{attribute 'linkalways'} 
{attribute 'no_explicit_call' := 'This FB is a CLASS and must be accessed using methods or properties'}
{attribute 'enable_dynamic_creation'}
FUNCTION_BLOCK _DT EXTENDS DatatypeBase
VAR
	localData : DT;
	activeData : REFERENCE TO DT REF= localData;
END_VAR

PROPERTY PUBLIC Address : PVOID
GET
Address := ADR(activeData);
END_GET
END_PROPERTY

METHOD PUBLIC ClearReference
VAR_INPUT
END_VAR
activeData REF= localData;
END_METHOD

METHOD PUBLIC Clone : I_Datatype
VAR
    pClone : POINTER TO _DT;
END_VAR
pClone := __NEW(_DT(InitialValue := Value));
Clone := pClone^;
END_METHOD

METHOD FB_init : BOOL
VAR_INPUT
	bInitRetains : BOOL; // if TRUE, the retain variables are initialized (warm start / cold start)
	bInCopyCode : BOOL;  // if TRUE, the instance afterwards gets moved WORDo the copy code (online change)
	InitialValue : DT;
END_VAR
localData := InitialValue;
END_METHOD

PROPERTY PUBLIC IecType : T_MAXSTRING
GET
IecType := 'DT';
END_GET
END_PROPERTY

METHOD PUBLIC MakeReferenceTo
VAR_INPUT
	ReferenceTarget : REFERENCE TO DT;
END_VAR
activeData REF= ReferenceTarget;
END_METHOD

METHOD PUBLIC SerializeWith
VAR_INPUT
	Serializer : I_Serializer;
END_VAR
Serializer.AddDateTime(activeData);
END_METHOD

PROPERTY PUBLIC Size : UDINT
GET
Size := SIZEOF(activeData);
END_GET
END_PROPERTY

METHOD TryDeserializeFrom : BOOL
VAR_INPUT
	Deserializer : I_Deserializer;
	Feedback : I_DeserializerFeedback;
END_VAR
TryDeserializeFrom := Deserializer.TryGetDateTime(activeData, Feedback);
END_METHOD

METHOD TryMakeReferenceTo : BOOL
VAR_INPUT
	Target : I_Datatype;
END_VAR
VAR
	pTargetData : POINTER TO DT;
END_VAR
IF NOT (Target.IecType = IecType) THEN
	RETURN;
END_IF

pTargetData := Target.Address;
activeData REF= pTargetData^;
TryMakeReferenceTo := TRUE;
END_METHOD

PROPERTY PUBLIC Value : DT
GET
Value := activeData;
END_GET
SET
activeData := Value;
END_SET
END_PROPERTY

END_FUNCTION_BLOCK

(* stored: Version 1.1.0.1, ProductVersion 3.1.4024.12
   POU _DT: Id {5f0ed87a-efb3-0af3-3883-e19c081fdc00}, SpecialFunc None
   Folder Constructor: Id {29a57be8-9521-02ea-0210-43bf4e6f5595}
   Property Address: Id {01c07cd3-6ad8-0564-0c4b-2911104e3390}
   Get Get: Id {4c43ffa5-0c61-027d-3467-332c73ced3a6}
   Method ClearReference: Id {facc431e-3b24-02fc-2270-310f5a719454}
   Method Clone: Id {5f3d84b8-a743-0597-324d-f0078728fbc7}
   Method FB_init: Id {a1a061fc-f3bd-057e-3e6f-b4a094d0b439}
   Property IecType: Id {5a60c3be-49e4-0bea-33b1-0c3ea06f8245}
   Get Get: Id {0bd9b606-ce90-0f09-3b04-07eb42523072}
   Method MakeReferenceTo: Id {cfaca68c-b5d9-0493-2bd5-08d57f7cf5c8}
   Method SerializeWith: Id {058b9483-f6fd-0db0-2f66-9967c26a5006}
   Property Size: Id {cf76693d-be61-0e6e-3cc5-cf07be7c91e4}
   Get Get: Id {87f63fd4-7fdb-06bf-28a4-92e806c3a9bb}
   Method TryDeserializeFrom: Id {c75775d3-2c3b-0353-23e3-1021ac167e6e}
   Method TryMakeReferenceTo: Id {5fbf191e-4728-0e31-14e3-de5ad17311b9}
   Property Value: Id {6dd914c3-1cd0-0085-00dc-d904ef41b507}
   Get Get: Id {feb495ac-5dac-0226-0aea-ab91655ec80e}
   Set Set: Id {8dc0cdfa-fb57-068d-37ee-bac3682a7e7d} *)
